// TIA Portal V18 export
// export: Created 2026-01-09T11:31:54.1359349Z, ExportSetting WithDefaults, DisplayName Totally Integrated Automation Portal, DisplayVersion V18 Update 5, DisplayName TIA Portal Openness, DisplayVersion V18 Update 5, DisplayName TIA Portal Teamcenter Gateway, DisplayVersion V18, DisplayName TIA Portal Version Control Interface, DisplayVersion V18, DisplayName SINAMICS Startdrive Advanced, DisplayVersion V18 SP2 Update 1, DisplayName SINAMICS Startdrive G110M, G120, G120C, G120D, G120P, G115D, DisplayVersion V18 SP2 Update 1, DisplayName SINAMICS Startdrive G130, G150, S120, S150, SINAMICS MV, S210, G220, S200, DisplayVersion V18 SP2 Update 1, DisplayName STEP 7 Professional, DisplayVersion V18 Update 5, DisplayName STEP 7 Safety, DisplayVersion V18, DisplayName WinCC Professional, DisplayVersion V18 Update 5
TagTable "StationStatus"
  Status_A1TableScanStatus : Int  (PLC tag AutoProcessControl.Status.A1TableScan.Status, CPU S71500-2PN_TP700, 1 s)
  Status_B1Press_Status : Int  (PLC tag AutoProcessControl.Status.B1Press.Status, CPU S71500-2PN_TP700, 1 s)
  Status_B2Press_Status : Int  (PLC tag AutoProcessControl.Status.B2Press.Status, CPU S71500-2PN_TP700, 1 s)
  Status_C_Glue_Status : Int  (PLC tag AutoProcessControl.Status.CGlueing.Status, CPU S71500-2PN_TP700, 1 s)
  Status_ENG_1_Status : Int  (PLC tag AutoProcessControl.Status.ENG_1.Status, CPU S71500-2PN_TP700, 1 s)
  Status_ENG_2_Status : Int  (PLC tag AutoProcessControl.Status.ENG_2.Status, CPU S71500-2PN_TP700, 1 s)
  Status_FRobot_1_Status : Int  (PLC tag AutoProcessControl.Status.FRobot_1.Status, CPU S71500-2PN_TP700, 1 s)
  Status_FRobot_2_Status : Int  (PLC tag AutoProcessControl.Status.FRobot_2.Status, CPU S71500-2PN_TP700, 1 s)
  Status_FRobot_3_Status : Int  (PLC tag AutoProcessControl.Status.FRobot_3.Status, CPU S71500-2PN_TP700, 1 s)
  StationStatusH : Int  (PLC tag AutoProcessControl.Status.HShaftLifting.Status, CPU S71500-2PN_TP700, 1 s)
  StationStatusJ : Int  (PLC tag AutoProcessControl.Status.JMagnetLifting.Status, CPU S71500-2PN_TP700, 1 s)
  StationStatusK : Int  (PLC tag AutoProcessControl.Status.KReserveLifting.Status, CPU S71500-2PN_TP700, 1 s)
  HMI_ESTOP : Bool  (PLC tag ST10_SysInput.HMI_Button.E-Stop, CPU S71500-2PN_TP700, 1 s)
  ESTOP_PB1 : Bool  (PLC tag ST10_SysInput.iE-StopPB[1], CPU S71500-2PN_TP700, 1 s)
  ESTOP_PB2 : Bool  (PLC tag ST10_SysInput.iE-StopPB[2], CPU S71500-2PN_TP700, 1 s)
  ESTOP_PB3 : Bool  (PLC tag ST10_SysInput.iE-StopPB[3], CPU S71500-2PN_TP700, 1 s)
  ESTOP_PB4 : Bool  (PLC tag ST10_SysInput.iE-StopPB[4], CPU S71500-2PN_TP700, 1 s)
  ESTOP_PB5 : Bool  (PLC tag ST10_SysInput.iE-StopPB[5], CPU S71500-2PN_TP700, 1 s)
  ESTOP_PB6 : Bool  (PLC tag ST10_SysInput.iE-StopPB[6], CPU S71500-2PN_TP700, 1 s)
  ESTOP_PB7 : Bool  (PLC tag ST10_SysInput.iE-StopPB[7], CPU S71500-2PN_TP700, 1 s)
  ESTOP_PB8 : Bool  (PLC tag ST10_SysInput.iE-StopPB[8], CPU S71500-2PN_TP700, 1 s)
  ESTOP_PB9 : Bool  (PLC tag ST10_SysInput.iE-StopPB[9], CPU S71500-2PN_TP700, 1 s)
  ESTOP_PB10 : Bool  (PLC tag ST10_SysInput.iE-StopPB[10], CPU S71500-2PN_TP700, 1 s)
  ESTOP_PB11 : Bool  (PLC tag ST10_SysInput.iE-StopPB[11], CPU S71500-2PN_TP700, 1 s)
  ESTOP_PB12 : Bool  (PLC tag ST10_SysInput.iE-StopPB[12], CPU S71500-2PN_TP700, 1 s)
  Status_A2TableScanStatus : Int  (PLC tag AutoProcessControl.Status.A2TableScan.Status, CPU S71500-2PN_TP700, 1 s)
  StationStatusL : Int  (PLC tag AutoProcessControl.Status.LUnloadingTrans.Status, CPU S71500-2PN_TP700, 1 s)
  Status_Solidify_Status : Int  (PLC tag AutoProcessControl.Status.Solidify.Status, CPU S71500-2PN_TP700, 1 s)
